{attribute 'linkalways'} 
{attribute 'no_explicit_call' := 'This FB is a CLASS and must be accessed using methods or properties'}
{attribute 'enable_dynamic_creation'}
FUNCTION_BLOCK Node_F_VN_ConvertColorSpace EXTENDS Node
VAR
	ipSrcImage : _ITcVnImage;
    ipDestImage : _ITcVnImage;
    eTransform : _ETcVnColorSpaceTransform(ETcVnColorSpaceTransform.TCVN_CST_RGBA_TO_RGB);
    hrPrev : _HRESULT(S_OK);
	hresult : _HRESULT(S_OK);
END_VAR

METHOD PUBLIC  Clone : I_Node
VAR
	pNode : POINTER TO Node_F_VN_ConvertColorSpace;
END_VAR
pNode := __NEW(Node_F_VN_ConvertColorSpace);
Clone := pNode^;
END_METHOD

METHOD FB_init : BOOL
VAR_INPUT
	bInitRetains : BOOL; // if TRUE, the retain variables are initialized (warm start / cold start)
	bInCopyCode : BOOL;  // if TRUE, the instance afterwards gets moved into the copy code (online change)
END_VAR
AddInput('ipSrcImage', ipSrcImage);
AddInput('hrPrev', hrPrev);
AddOutput('ipDestImage', ipDestImage);
AddOutput('hresult',hresult);
AddParameter('eTransform', eTransform);
END_METHOD

METHOD PROTECTED  OnExecute : HRESULT
hresult.Value := F_VN_ConvertColorSpace(
	ipSrcImage   := ipSrcImage.Value, 
	ipDestImage:= ipDestImage.Value, 
	eTransform := eTransform.Value, 
	hrPrev := hrPrev.Value);
END_METHOD

END_FUNCTION_BLOCK

(* stored: Version 1.1.0.1, ProductVersion 3.1.4024.13
   POU Node_F_VN_ConvertColorSpace: Id {be1766e7-e6ea-06a3-0c0f-bb81e570288e}, SpecialFunc None
   Folder Constructor: Id {b65dc154-1ac1-03c4-346d-19e138c362f3}
   Method Clone: Id {183571d5-5395-0956-1776-d98504f3987a}
   Method FB_init: Id {e16bba1c-071e-065e-38b1-878340e733eb}
   Method OnExecute: Id {0faaad2b-dd3f-0d95-2f39-1f13ef681cd5} *)
